// TIA Portal project "Lezione2_CorsoBase" (V19)

(* hardware
DEVICE "S7-1200 station_1"  S7-1200 Station
   slot 0: "Rack_0"  S7-1200 Rack  Rack  V1.0
   slot 1: "PLC_1"  CPU 1214C AC/DC/Rly  6ES7 214-1BG40-0XB0  V4.1
*)

// ===== PLC "PLC_1"  CPU 1214C AC/DC/Rly =====

VAR_GLOBAL   // PLC tag table "Default tag table"
   "PulsanteEmergenza" AT %I0.0 : Bool;
   "PulsanteStop" AT %I0.1 : Bool;
   "TermicaMotore" AT %I0.2 : Bool;
   "StartAvanti" AT %I0.3 : Bool;
   "StartIndietro" AT %I0.4 : Bool;
   "ResetAllarmi" AT %I0.5 : Bool;
   "ResetConteggio" AT %I0.6 : Bool;
   "MotoreAvanti" AT %Q0.0 : Bool;
   "MotoreIndietro" AT %Q0.1 : Bool;
   "LampadaVerde" AT %Q0.2 : Bool;
   "LampadaGialla" AT %Q0.3 : Bool;
   "LampadaRossa" AT %Q0.4 : Bool;
END_VAR

DATA_BLOCK "Motore1"   // DB1
{ S7_Optimized_Access := 'TRUE' }
VERSION : 0.1
// stored: InstanceOfName Motore
"Motore"
BEGIN
END_DATA_BLOCK

DATA_BLOCK "Motore_ST_2"   // DB2
{ S7_Optimized_Access := 'TRUE' }
VERSION : 0.1
// stored: InstanceOfName Motore_ST
"Motore_ST"
BEGIN
END_DATA_BLOCK

FUNCTION_BLOCK "Motore"   // FB1, LAD
{ S7_Optimized_Access := 'TRUE' }
VERSION : 0.1
   VAR_INPUT
      StartAvanti : Bool;
      StartIndietro : Bool;
      Stop : Bool;
      Termica : Bool;
      Emergenza : Bool;
      ResetAllarme : Bool;
      ResetConteggio : Bool;
   END_VAR
   VAR_OUTPUT
      MotoreAvanti : Bool;
      MotoreIndietro : Bool;
      StatoAttuale : Int;
   END_VAR
   VAR
      AllarmeAttivo : Bool;
   END_VAR
   VAR CONSTANT
      STATO_FERMO : Int := 0;
      STATO_AVANTI : Int := 100;
      STATO_INDIETRO : Int := 200;
      STATO_EMERGENZA : Int := 1000;
   END_VAR
   VAR_TEMP   // added for the SCL form of the ladder/FBD networks
      _w1 : Bool;
   END_VAR
BEGIN

REGION Network 1
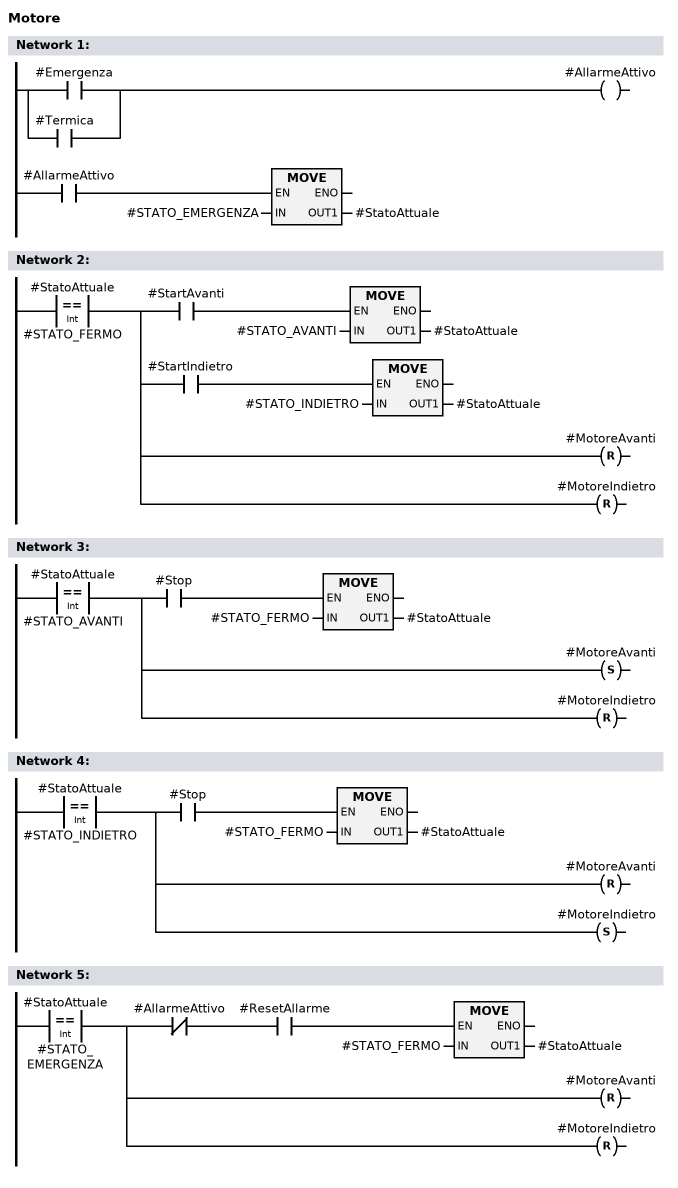
   RUNG wire#powerrail
      Contact( #Emergenza )
      wire#w1
      Coil( #AllarmeAttivo )
   END_RUNG
   RUNG wire#powerrail
      Contact( #Termica )
   END_RUNG wire#w1
   RUNG wire#powerrail
      Contact( #AllarmeAttivo )
      Move(in := #STATO_EMERGENZA, out1 => #StatoAttuale)
   END_RUNG
   // the same network as SCL:
   #AllarmeAttivo := #Emergenza OR #Termica;
   IF #AllarmeAttivo THEN #StatoAttuale := #STATO_EMERGENZA; END_IF;
END_REGION

REGION Network 2
   RUNG wire#powerrail
      { S7_Templates := "SrcType := Int" } EQ_Contact(in1 := #StatoAttuale, in2 := #STATO_FERMO)
      wire#w1
      Contact( #StartAvanti )
      Move(in := #STATO_AVANTI, out1 => #StatoAttuale)
   END_RUNG
   RUNG wire#w1
      Contact( #StartIndietro )
      Move(in := #STATO_INDIETRO, out1 => #StatoAttuale)
   END_RUNG
   RUNG wire#w1
      R_Coil( #MotoreAvanti )
   END_RUNG
   RUNG wire#w1
      R_Coil( #MotoreIndietro )
   END_RUNG
   // the same network as SCL:
   #_w1 := #StatoAttuale = #STATO_FERMO;
   IF #_w1 AND #StartAvanti THEN #StatoAttuale := #STATO_AVANTI; END_IF;
   IF #_w1 AND #StartIndietro THEN #StatoAttuale := #STATO_INDIETRO; END_IF;
   IF #_w1 THEN
       #MotoreAvanti := FALSE;
       #MotoreIndietro := FALSE;
   END_IF;
END_REGION

REGION Network 3
   RUNG wire#powerrail
      { S7_Templates := "SrcType := Int" } EQ_Contact(in1 := #StatoAttuale, in2 := #STATO_AVANTI)
      wire#w1
      Contact( #Stop )
      Move(in := #STATO_FERMO, out1 => #StatoAttuale)
   END_RUNG
   RUNG wire#w1
      S_Coil( #MotoreAvanti )
   END_RUNG
   RUNG wire#w1
      R_Coil( #MotoreIndietro )
   END_RUNG
   // the same network as SCL:
   #_w1 := #StatoAttuale = #STATO_AVANTI;
   IF #_w1 AND #Stop THEN #StatoAttuale := #STATO_FERMO; END_IF;
   IF #_w1 THEN
       #MotoreAvanti := TRUE;
       #MotoreIndietro := FALSE;
   END_IF;
END_REGION

REGION Network 4
   RUNG wire#powerrail
      { S7_Templates := "SrcType := Int" } EQ_Contact(in1 := #StatoAttuale, in2 := #STATO_INDIETRO)
      wire#w1
      Contact( #Stop )
      Move(in := #STATO_FERMO, out1 => #StatoAttuale)
   END_RUNG
   RUNG wire#w1
      R_Coil( #MotoreAvanti )
   END_RUNG
   RUNG wire#w1
      S_Coil( #MotoreIndietro )
   END_RUNG
   // the same network as SCL:
   #_w1 := #StatoAttuale = #STATO_INDIETRO;
   IF #_w1 AND #Stop THEN #StatoAttuale := #STATO_FERMO; END_IF;
   IF #_w1 THEN
       #MotoreAvanti := FALSE;
       #MotoreIndietro := TRUE;
   END_IF;
END_REGION

REGION Network 5
   RUNG wire#powerrail
      { S7_Templates := "SrcType := Int" } EQ_Contact(in1 := #StatoAttuale, in2 := #STATO_EMERGENZA)
      wire#w1
      I_Contact( #AllarmeAttivo )
      Contact( #ResetAllarme )
      Move(in := #STATO_FERMO, out1 => #StatoAttuale)
   END_RUNG
   RUNG wire#w1
      R_Coil( #MotoreAvanti )
   END_RUNG
   RUNG wire#w1
      R_Coil( #MotoreIndietro )
   END_RUNG
   // the same network as SCL:
   #_w1 := #StatoAttuale = #STATO_EMERGENZA;
   IF #_w1 AND NOT #AllarmeAttivo AND #ResetAllarme THEN #StatoAttuale := #STATO_FERMO; END_IF;
   IF #_w1 THEN
       #MotoreAvanti := FALSE;
       #MotoreIndietro := FALSE;
   END_IF;
END_REGION
END_FUNCTION_BLOCK

FUNCTION_BLOCK "Motore_ST"   // FB2, SCL
{ S7_Optimized_Access := 'TRUE' }
VERSION : 0.1
   VAR_INPUT
      StartAvanti : Bool;
      StartIndietro : Bool;
      Stop : Bool;
      Termica : Bool;
      Emergenza : Bool;
      ResetAllarme : Bool;
      ResetConteggio : Bool;
   END_VAR
   VAR_OUTPUT
      MotoreAvanti : Bool;
      MotoreIndietro : Bool;
      StatoAttuale : Int;
   END_VAR
   VAR
      AllarmeAttivo : Bool;
   END_VAR
   VAR CONSTANT
      STATO_FERMO : Int := 0;
      STATO_AVANTI : Int := 100;
      STATO_INDIETRO : Int := 200;
      STATO_EMERGENZA : Int := 1000;
   END_VAR
BEGIN

   #AllarmeAttivo := #Emergenza OR #Termica;
   IF #AllarmeAttivo THEN
       #StatoAttuale := #STATO_EMERGENZA;
   END_IF;



   CASE #StatoAttuale OF
       #STATO_FERMO:

           #MotoreAvanti   := FALSE;
           #MotoreIndietro := FALSE;

           IF #StartAvanti THEN
               #StatoAttuale := #STATO_AVANTI;
           END_IF;


           IF #StartIndietro THEN
               #StatoAttuale := #STATO_INDIETRO;
           END_IF;


       #STATO_AVANTI:

           #MotoreAvanti   := TRUE;
           #MotoreIndietro := FALSE;

           IF #Stop THEN
               #StatoAttuale := #STATO_FERMO;
           END_IF



       #STATO_INDIETRO:

           #MotoreAvanti   := FALSE;
           #MotoreIndietro := TRUE;

           IF #Stop THEN
               #StatoAttuale := #STATO_FERMO;
           END_IF


       #STATO_EMERGENZA:

           #MotoreAvanti   := FALSE;
           #MotoreIndietro := FALSE;

           IF NOT #AllarmeAttivo AND #ResetAllarme THEN
               #StatoAttuale := #STATO_FERMO;
           END_IF;


   END_CASE;
END_FUNCTION_BLOCK

ORGANIZATION_BLOCK "Main"   // OB1, LAD, ProgramCycle
TITLE = "Main Program Sweep (Cycle)"
{ S7_Optimized_Access := 'TRUE' }
VERSION : 0.1
   VAR_INPUT
      Initial_Call : Bool;   // Initial call of this OB
      Remanence : Bool;   // =True, if remanent data are available
   END_VAR
BEGIN

REGION Network 1
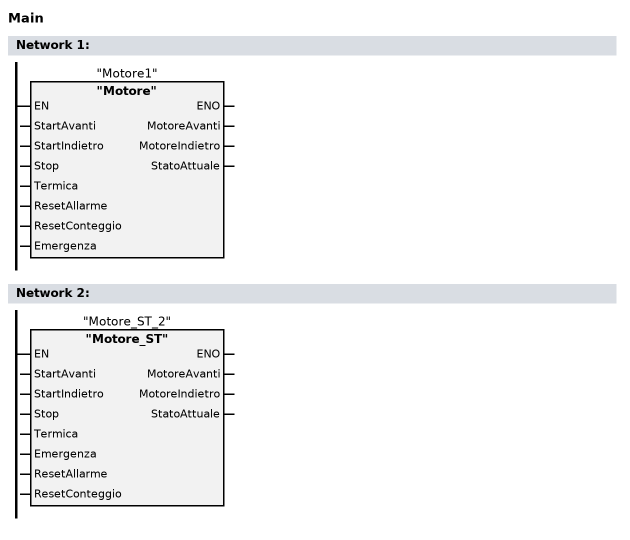
   RUNG wire#powerrail
      "Motore1"(StartAvanti :=, StartIndietro :=, Stop :=, Termica :=, ResetAllarme :=, ResetConteggio :=, Emergenza :=, MotoreAvanti =>, MotoreIndietro =>, StatoAttuale =>)
   END_RUNG
   // the same network as SCL:
   "Motore1"();   // "Motore"
END_REGION

REGION Network 2
   RUNG wire#powerrail
      "Motore_ST_2"(StartAvanti :=, StartIndietro :=, Stop :=, Termica :=, Emergenza :=, ResetAllarme :=, ResetConteggio :=, MotoreAvanti =>, MotoreIndietro =>, StatoAttuale =>)
   END_RUNG
   // the same network as SCL:
   "Motore_ST_2"();   // "Motore_ST"
END_REGION
END_ORGANIZATION_BLOCK